Fanuc TP program (LS listing): ground_truth.ls

/PROG  TOR_XL_LEARN_V3
/ATTR
OWNER		= MNEDITOR;
COMMENT		= "WeldPRO Auto-Gen";
PROG_SIZE	= 7125;
CREATE		= DATE 26-07-30  TIME 15:09:28;
MODIFIED	= DATE 26-07-30  TIME 15:41:30;
FILE_NAME	= TOR_XL_L;
VERSION		= 0;
LINE_COUNT	= 113;
MEMORY_SIZE	= 7445;
PROTECT		= READ_WRITE;
TCD:  STACK_SIZE	= 0,
      TASK_PRIORITY	= 50,
      TIME_SLICE	= 0,
      BUSY_LAMP_OFF	= 0,
      ABORT_REQUEST	= 0,
      PAUSE_REQUEST	= 0;
DEFAULT_GROUP	= 1,*,*,*,*;
CONTROL_CODE	= 00000000 00000000;
/APPL
/MN
   1:  !WeldPRO Auto-Generated TPP ;
   2:  !TOR_XL_2026, TOR_xl_2907 ;
   3:   ;
   4:  UFRAME_NUM=2 ;
   5:  UTOOL_NUM=2 ;
   6:  !Feature Approach ;
   7:J P[1]{
   GP1:
	UF : 2, UT : 2,		CONFIG : 'F D T, 0, 0, 0',
	X =   924.335  mm,	Y =   780.986  mm,	Z =  -268.284  mm,
	W =  -106.495 deg,	P =   -15.000 deg,	R =    94.234 deg
};
P[2]{
   GP1:
	UF : 2, UT : 2,		CONFIG : 'F D T, 0, 0, 0',
	X =  1018.715  mm,	Y =   787.224  mm,	Z =  -235.231  mm,
	W =  -106.492 deg,	P =   -15.098 deg,	R =    90.372 deg
};
P[3]{
   GP1:
	UF : 2, UT : 2,		CONFIG : 'F D T, 0, 0, 0',
	X =  1020.495  mm,	Y =   807.281  mm,	Z =  -235.073  mm,
	W =  -106.456 deg,	P =   -15.335 deg,	R =    80.815 deg
};
P[4]{
   GP1:
	UF : 2, UT : 2,		CONFIG : 'F D T, 0, 0, 0',
	X =  1022.247  mm,	Y =   817.408  mm,	Z =  -235.756  mm,
	W =  -106.423 deg,	P =   -15.450 deg,	R =    76.090 deg
};
P[5]{
   GP1:
	UF : 2, UT : 2,		CONFIG : 'F D T, 0, 0, 0',
	X =  1025.517  mm,	Y =   826.963  mm,	Z =  -235.844  mm,
	W =  -106.378 deg,	P =   -15.565 deg,	R =    71.217 deg
};
P[6]{
   GP1:
	UF : 2, UT : 2,		CONFIG : 'F D T, 0, 0, 0',
	X =  1029.053  mm,	Y =   836.370  mm,	Z =  -235.876  mm,
	W =  -106.322 deg,	P =   -15.679 deg,	R =    66.207 deg
};
P[7]{
   GP1:
	UF : 2, UT : 2,		CONFIG : 'F D T, 0, 0, 0',
	X =  1033.689  mm,	Y =   845.357  mm,	Z =  -236.189  mm,
	W =  -106.254 deg,	P =   -15.791 deg,	R =    61.015 deg
};
P[8]{
   GP1:
	UF : 2, UT : 2,		CONFIG : 'F D T, 0, 0, 0',
	X =  1038.830  mm,	Y =   853.927  mm,	Z =  -236.142  mm,
	W =  -106.177 deg,	P =   -15.894 deg,	R =    55.979 deg
};
P[9]{
   GP1:
	UF : 2, UT : 2,		CONFIG : 'F D T, 0, 0, 0',
	X =  1045.034  mm,	Y =   861.671  mm,	Z =  -235.917  mm,
	W =  -106.096 deg,	P =   -15.986 deg,	R =    51.162 deg
};
P[10]{
   GP1:
	UF : 2, UT : 2,		CONFIG : 'F D T, 0, 0, 0',
	X =  1051.595  mm,	Y =   869.013  mm,	Z =  -235.579  mm,
	W =  -106.012 deg,	P =   -16.066 deg,	R =    46.632 deg
};
P[11]{
   GP1:
	UF : 2, UT : 2,		CONFIG : 'F D T, 0, 0, 0',
	X =  1058.405  mm,	Y =   876.388  mm,	Z =  -235.876  mm,
	W =  -105.919 deg,	P =   -16.142 deg,	R =    41.952 deg
};
P[12]{
   GP1:
	UF : 2, UT : 2,		CONFIG : 'F D T, 0, 0, 0',
	X =  1066.182  mm,	Y =   882.960  mm,	Z =  -236.508  mm,
	W =  -105.870 deg,	P =   -16.177 deg,	R =    39.609 deg
};
P[13]{
   GP1:
	UF : 2, UT : 2,		CONFIG : 'F D T, 0, 0, 0',
	X =  1074.017  mm,	Y =   888.320  mm,	Z =  -234.957  mm,
	W =  -105.777 deg,	P =   -16.235 deg,	R =    35.365 deg
};
P[14]{
   GP1:
	UF : 2, UT : 2,		CONFIG : 'F D T, 0, 0, 0',
	X =  1082.402  mm,	Y =   893.773  mm,	Z =  -235.312  mm,
	W =  -105.677 deg,	P =   -16.289 deg,	R =    30.964 deg
};
P[15]{
   GP1:
	UF : 2, UT : 2,		CONFIG : 'F D T, 0, 0, 0',
	X =  1091.030  mm,	Y =   899.008  mm,	Z =  -235.877  mm,
	W =  -105.579 deg,	P =   -16.333 deg,	R =    26.830 deg
};
P[16]{
   GP1:
	UF : 2, UT : 2,		CONFIG : 'F D T, 0, 0, 0',
	X =  1100.156  mm,	Y =   902.452  mm,	Z =  -235.103  mm,
	W =  -105.537 deg,	P =   -16.344 deg,	R =    25.018 deg
};
P[17]{
   GP1:
	UF : 2, UT : 2,		CONFIG : 'F D T, 0, 0, 0',
	X =  1109.917  mm,	Y =   906.637  mm,	Z =  -236.186  mm,
	W =  -116.027 deg,	P =   -16.063 deg,	R =    30.267 deg
};
P[18]{
   GP1:
	UF : 2, UT : 2,		CONFIG : 'F D T, 0, 0, 0',
	X =  1118.157  mm,	Y =   911.916  mm,	Z =  -235.088  mm,
	W =  -126.877 deg,	P =   -15.356 deg,	R =    25.893 deg
};
P[19]{
   GP1:
	UF : 2, UT : 2,		CONFIG : 'F D T, 0, 0, 0',
	X =  1124.146  mm,	Y =   914.820  mm,	Z =  -228.920  mm,
	W =  -119.393 deg,	P =   -15.981 deg,	R =    16.221 deg
};
P[20]{
   GP1:
	UF : 2, UT : 2,		CONFIG : 'F D T, 0, 0, 0',
	X =  1129.948  mm,	Y =   917.746  mm,	Z =  -222.103  mm,
	W =  -115.329 deg,	P =   -16.208 deg,	R =    11.788 deg
};
P[21]{
   GP1:
	UF : 2, UT : 2,		CONFIG : 'F D T, 0, 0, 0',
	X =  1135.715  mm,	Y =   919.222  mm,	Z =  -213.573  mm,
	W =  -112.639 deg,	P =   -16.315 deg,	R =     9.714 deg
};
P[22]{
   GP1:
	UF : 2, UT : 2,		CONFIG : 'F D T, 0, 0, 0',
	X =  1142.436  mm,	Y =   921.368  mm,	Z =  -205.545  mm,
	W =  -110.015 deg,	P =   -16.386 deg,	R =     9.649 deg
};
P[23]{
   GP1:
	UF : 2, UT : 2,		CONFIG : 'F D T, 0, 0, 0',
	X =  1147.023  mm,	Y =   921.905  mm,	Z =  -202.145  mm,
	W =  -108.552 deg,	P =   -16.418 deg,	R =     8.950 deg
};
P[24]{
   GP1:
	UF : 2, UT : 2,		CONFIG : 'F D T, 0, 0, 0',
	X =  1160.278  mm,	Y =   924.170  mm,	Z =  -197.796  mm,
	W =  -105.409 deg,	P =   -16.443 deg,	R =     6.805 deg
};
P[25]{
   GP1:
	UF : 2, UT : 2,		CONFIG : 'F D T, 0, 0, 0',
	X =  1169.888  mm,	Y =   925.126  mm,	Z =  -196.732  mm,
	W =  -104.866 deg,	P =   -16.444 deg,	R =     5.597 deg
};
P[26]{
   GP1:
	UF : 2, UT : 2,		CONFIG : 'F D T, 0, 0, 0',
	X =  1179.662  mm,	Y =   926.011  mm,	Z =  -196.715  mm,
	W =  -104.887 deg,	P =   -16.444 deg,	R =     3.523 deg
};
P[27]{
   GP1:
	UF : 2, UT : 2,		CONFIG : 'F D T, 0, 0, 0',
	X =  1189.383  mm,	Y =   926.437  mm,	Z =  -196.950  mm,
	W =  -104.930 deg,	P =   -16.439 deg,	R =     -.729 deg
};
P[28]{
   GP1:
	UF : 2, UT : 2,		CONFIG : 'F D T, 0, 0, 0',
	X =  1199.044  mm,	Y =   925.579  mm,	Z =  -197.248  mm,
	W =  -104.979 deg,	P =   -16.424 deg,	R =    -5.541 deg
};
P[29]{
   GP1:
	UF : 2, UT : 2,		CONFIG : 'F D T, 0, 0, 0',
	X =  1208.438  mm,	Y =   924.247  mm,	Z =  -196.868  mm,
	W =  -105.028 deg,	P =   -16.400 deg,	R =   -10.259 deg
};
P[30]{
   GP1:
	UF : 2, UT : 2,		CONFIG : 'F D T, 0, 0, 0',
	X =  1218.046  mm,	Y =   922.651  mm,	Z =  -197.246  mm,
	W =  -105.070 deg,	P =   -16.371 deg,	R =   -14.490 deg
};
P[31]{
   GP1:
	UF : 2, UT : 2,		CONFIG : 'F D T, 0, 0, 0',
	X =  1227.367  mm,	Y =   919.386  mm,	Z =  -197.752  mm,
	W =  -105.112 deg,	P =   -16.334 deg,	R =   -18.515 deg
};
P[32]{
   GP1:
	UF : 2, UT : 2,		CONFIG : 'F D T, 0, 0, 0',
	X =  1236.641  mm,	Y =   916.419  mm,	Z =  -198.075  mm,
	W =  -105.158 deg,	P =   -16.285 deg,	R =   -23.051 deg
};
P[33]{
   GP1:
	UF : 2, UT : 2,		CONFIG : 'F D T, 0, 0, 0',
	X =  1245.126  mm,	Y =   912.315  mm,	Z =  -197.759  mm,
	W =  -105.219 deg,	P =   -16.204 deg,	R =   -29.417 deg
};
P[34]{
   GP1:
	UF : 2, UT : 2,		CONFIG : 'F D T, 0, 0, 0',
	X =  1252.682  mm,	Y =   907.045  mm,	Z =  -197.652  mm,
	W =  -105.311 deg,	P =   -16.047 deg,	R =   -39.415 deg
};
P[35]{
   GP1:
	UF : 2, UT : 2,		CONFIG : 'F D T, 0, 0, 0',
	X =  1260.941  mm,	Y =   901.305  mm,	Z =  -197.740  mm,
	W =  -105.307 deg,	P =   -16.055 deg,	R =   -38.974 deg
};
P[36]{
   GP1:
	UF : 2, UT : 2,		CONFIG : 'F D T, 0, 0, 0',
	X =  1267.955  mm,	Y =   894.273  mm,	Z =  -197.409  mm,
	W =  -105.302 deg,	P =   -16.063 deg,	R =   -38.625 deg
};
P[37]{
   GP1:
	UF : 2, UT : 2,		CONFIG : 'F D T, 0, 0, 0',
	X =  1276.534  mm,	Y =   889.263  mm,	Z =  -197.995  mm,
	W =  -105.469 deg,	P =   -15.944 deg,	R =   -44.976 deg
};
P[38]{
   GP1:
	UF : 2, UT : 2,		CONFIG : 'F D T, 0, 0, 0',
	X =  1283.155  mm,	Y =   882.295  mm,	Z =  -197.847  mm,
	W =  -105.661 deg,	P =   -15.890 deg,	R =   -47.714 deg
};
P[39]{
   GP1:
	UF : 2, UT : 2,		CONFIG : 'F D T, 0, 0, 0',
	X =  1289.852  mm,	Y =   875.249  mm,	Z =  -198.875  mm,
	W =  -106.210 deg,	P =   -15.792 deg,	R =   -52.259 deg
};
P[40]{
   GP1:
	UF : 2, UT : 2,		CONFIG : 'F D T, 0, 0, 0',
	X =  1296.112  mm,	Y =   867.768  mm,	Z =  -200.273  mm,
	W =  -106.927 deg,	P =   -15.688 deg,	R =   -56.663 deg
};
P[41]{
   GP1:
	UF : 2, UT : 2,		CONFIG : 'F D T, 0, 0, 0',
	X =  1301.774  mm,	Y =   859.713  mm,	Z =  -202.128  mm,
	W =  -107.603 deg,	P =   -15.597 deg,	R =   -60.243 deg
};
P[42]{
   GP1:
	UF : 2, UT : 2,		CONFIG : 'F D T, 0, 0, 0',
	X =  1306.016  mm,	Y =   850.984  mm,	Z =  -203.650  mm,
	W =  -108.271 deg,	P =   -15.504 deg,	R =   -63.685 deg
};
P[43]{
   GP1:
	UF : 2, UT : 2,		CONFIG : 'F D T, 0, 0, 0',
	X =  1309.573  mm,	Y =   842.117  mm,	Z =  -204.775  mm,
	W =  -109.144 deg,	P =   -15.377 deg,	R =   -68.203 deg
};
P[44]{
   GP1:
	UF : 2, UT : 2,		CONFIG : 'F D T, 0, 0, 0',
	X =  1313.875  mm,	Y =   833.270  mm,	Z =  -206.451  mm,
	W =  -109.899 deg,	P =   -15.253 deg,	R =   -72.505 deg
};
P[45]{
   GP1:
	UF : 2, UT : 2,		CONFIG : 'F D T, 0, 0, 0',
	X =  1317.383  mm,	Y =   823.850  mm,	Z =  -208.446  mm,
	W =  -110.273 deg,	P =   -15.181 deg,	R =   -74.981 deg
};
P[46]{
   GP1:
	UF : 2, UT : 2,		CONFIG : 'F D T, 0, 0, 0',
	X =  1319.294  mm,	Y =   814.046  mm,	Z =  -209.598  mm,
	W =  -110.635 deg,	P =   -14.305 deg,	R =   -78.232 deg
};
P[47]{
   GP1:
	UF : 2, UT : 2,		CONFIG : 'F D T, 0, 0, 0',
	X =  1321.222  mm,	Y =   804.155  mm,	Z =  -210.895  mm,
	W =  -111.054 deg,	P =   -14.769 deg,	R =   -83.164 deg
};
P[48]{
   GP1:
	UF : 2, UT : 2,		CONFIG : 'F D T, 0, 0, 0',
	X =  1322.108  mm,	Y =   794.074  mm,	Z =  -211.690  mm,
	W =  -111.190 deg,	P =   -15.305 deg,	R =   -88.308 deg
};
P[49]{
   GP1:
	UF : 2, UT : 2,		CONFIG : 'F D T, 0, 0, 0',
	X =  1322.417  mm,	Y =   783.924  mm,	Z =  -211.983  mm,
	W =  -111.129 deg,	P =   -15.645 deg,	R =   -91.614 deg
};
P[50]{
   GP1:
	UF : 2, UT : 2,		CONFIG : 'F D T, 0, 0, 0',
	X =  1321.632  mm,	Y =   773.848  mm,	Z =  -211.329  mm,
	W =  -110.761 deg,	P =   -14.624 deg,	R =   -96.574 deg
};
P[51]{
   GP1:
	UF : 2, UT : 2,		CONFIG : 'F D T, 0, 0, 0',
	X =  1320.812  mm,	Y =   763.757  mm,	Z =  -210.466  mm,
	W =  -110.276 deg,	P =   -14.535 deg,	R =  -100.836 deg
};
P[52]{
   GP1:
	UF : 2, UT : 2,		CONFIG : 'F D T, 0, 0, 0',
	X =  1318.396  mm,	Y =   754.196  mm,	Z =  -208.431  mm,
	W =  -109.635 deg,	P =   -14.447 deg,	R =  -105.265 deg
};
P[53]{
   GP1:
	UF : 2, UT : 2,		CONFIG : 'F D T, 0, 0, 0',
	X =  1315.879  mm,	Y =   744.538  mm,	Z =  -206.875  mm,
	W =  -109.083 deg,	P =   -14.382 deg,	R =  -108.625 deg
};
P[54]{
   GP1:
	UF : 2, UT : 2,		CONFIG : 'F D T, 0, 0, 0',
	X =  1312.567  mm,	Y =   735.090  mm,	Z =  -205.253  mm,
	W =  -108.349 deg,	P =   -14.302 deg,	R =  -112.873 deg
};
P[55]{
   GP1:
	UF : 2, UT : 2,		CONFIG : 'F D T, 0, 0, 0',
	X =  1308.961  mm,	Y =   725.703  mm,	Z =  -203.640  mm,
	W =  -107.748 deg,	P =   -14.239 deg,	R =  -116.265 deg
};
P[56]{
   GP1:
	UF : 2, UT : 2,		CONFIG : 'F D T, 0, 0, 0',
	X =  1305.001  mm,	Y =   716.454  mm,	Z =  -201.746  mm,
	W =  -106.927 deg,	P =   -14.148 deg,	R =  -121.193 deg
};
P[57]{
   GP1:
	UF : 2, UT : 2,		CONFIG : 'F D T, 0, 0, 0',
	X =  1299.050  mm,	Y =   708.363  mm,	Z =  -199.926  mm,
	W =  -106.269 deg,	P =   -14.066 deg,	R =  -125.698 deg
};
P[58]{
   GP1:
	UF : 2, UT : 2,		CONFIG : 'F D T, 0, 0, 0',
	X =  1293.324  mm,	Y =   700.186  mm,	Z =  -198.073  mm,
	W =  -105.781 deg,	P =   -13.988 deg,	R =  -130.143 deg
};
P[59]{
   GP1:
	UF : 2, UT : 2,		CONFIG : 'F D T, 0, 0, 0',
	X =  1286.894  mm,	Y =   692.340  mm,	Z =  -197.040  mm,
	W =  -105.529 deg,	P =   -13.914 deg,	R =  -134.519 deg
};
P[60]{
   GP1:
	UF : 2, UT : 2,		CONFIG : 'F D T, 0, 0, 0',
	X =  1279.894  mm,	Y =   684.848  mm,	Z =  -196.766  mm,
	W =  -105.437 deg,	P =   -13.849 deg,	R =  -138.629 deg
};
P[61]{
   GP1:
	UF : 2, UT : 2,		CONFIG : 'F D T, 0, 0, 0',
	X =  1272.475  mm,	Y =   678.006  mm,	Z =  -196.723  mm,
	W =  -105.429 deg,	P =   -13.831 deg,	R =  -139.837 deg
};
P[62]{
   GP1:
	UF : 2, UT : 2,		CONFIG : 'F D T, 0, 0, 0',
	X =  1265.641  mm,	Y =   670.880  mm,	Z =  -196.694  mm,
	W =  -105.443 deg,	P =   -13.863 deg,	R =  -137.727 deg
};
P[63]{
   GP1:
	UF : 2, UT : 2,		CONFIG : 'F D T, 0, 0, 0',
	X =  1257.021  mm,	Y =   664.482  mm,	Z =  -196.380  mm,
	W =  -105.373 deg,	P =   -13.729 deg,	R =  -147.436 deg
};
P[64]{
   GP1:
	UF : 2, UT : 2,		CONFIG : 'F D T, 0, 0, 0',
	X =  1247.675  mm,	Y =   659.504  mm,	Z =  -196.028  mm,
	W =  -105.298 deg,	P =   -13.637 deg,	R =  -156.529 deg
};
P[65]{
   GP1:
	UF : 2, UT : 2,		CONFIG : 'F D T, 0, 0, 0',
	X =  1238.718  mm,	Y =   654.671  mm,	Z =  -195.720  mm,
	W =  -105.277 deg,	P =   -13.618 deg,	R =  -158.976 deg
};
P[66]{
   GP1:
	UF : 2, UT : 2,		CONFIG : 'F D T, 0, 0, 0',
	X =  1229.052  mm,	Y =   650.811  mm,	Z =  -195.862  mm,
	W =  -105.241 deg,	P =   -13.592 deg,	R =  -162.969 deg
};
P[67]{
   GP1:
	UF : 2, UT : 2,		CONFIG : 'F D T, 0, 0, 0',
	X =  1219.160  mm,	Y =   648.075  mm,	Z =  -195.385  mm,
	W =  -105.203 deg,	P =   -13.573 deg,	R =  -167.022 deg
};
P[68]{
   GP1:
	UF : 2, UT : 2,		CONFIG : 'F D T, 0, 0, 0',
	X =  1208.921  mm,	Y =   646.203  mm,	Z =  -195.395  mm,
	W =  -105.159 deg,	P =   -13.560 deg,	R =  -171.569 deg
};
P[69]{
   GP1:
	UF : 2, UT : 2,		CONFIG : 'F D T, 0, 0, 0',
	X =  1198.642  mm,	Y =   645.785  mm,	Z =  -194.956  mm,
	W =  -105.113 deg,	P =   -13.556 deg,	R =  -176.312 deg
};
P[70]{
   GP1:
	UF : 2, UT : 2,		CONFIG : 'F D T, 0, 0, 0',
	X =  1188.344  mm,	Y =   645.393  mm,	Z =  -194.871  mm,
	W =  -105.068 deg,	P =   -13.561 deg,	R =   179.213 deg
};
P[71]{
   GP1:
	UF : 2, UT : 2,		CONFIG : 'F D T, 0, 0, 0',
	X =  1178.059  mm,	Y =   645.736  mm,	Z =  -195.139  mm,
	W =  -105.038 deg,	P =   -13.569 deg,	R =   176.231 deg
};
P[72]{
   GP1:
	UF : 2, UT : 2,		CONFIG : 'F D T, 0, 0, 0',
	X =  1167.871  mm,	Y =   646.652  mm,	Z =  -195.801  mm,
	W =  -105.207 deg,	P =   -13.572 deg,	R =   175.290 deg
};
P[73]{
   GP1:
	UF : 2, UT : 2,		CONFIG : 'F D T, 0, 0, 0',
	X =  1158.477  mm,	Y =   647.343  mm,	Z =  -195.653  mm,
	W =  -107.012 deg,	P =   -13.569 deg,	R =   174.537 deg
};
P[74]{
   GP1:
	UF : 2, UT : 2,		CONFIG : 'F D T, 0, 0, 0',
	X =  1149.730  mm,	Y =   648.837  mm,	Z =  -198.834  mm,
	W =  -109.414 deg,	P =   -13.538 deg,	R =   174.483 deg
};
P[75]{
   GP1:
	UF : 2, UT : 2,		CONFIG : 'F D T, 0, 0, 0',
	X =  1141.667  mm,	Y =   649.097  mm,	Z =  -206.147  mm,
	W =  -112.196 deg,	P =   -13.466 deg,	R =   175.323 deg
};
P[76]{
   GP1:
	UF : 2, UT : 2,		CONFIG : 'F D T, 0, 0, 0',
	X =  1135.547  mm,	Y =   650.958  mm,	Z =  -213.092  mm,
	W =  -114.872 deg,	P =   -13.369 deg,	R =   175.422 deg
};
P[77]{
   GP1:
	UF : 2, UT : 2,		CONFIG : 'F D T, 0, 0, 0',
	X =  1128.794  mm,	Y =   652.546  mm,	Z =  -221.828  mm,
	W =  -120.114 deg,	P =   -13.109 deg,	R =   172.293 deg
};
P[78]{
   GP1:
	UF : 2, UT : 2,		CONFIG : 'F D T, 0, 0, 0',
	X =  1122.507  mm,	Y =   656.297  mm,	Z =  -228.913  mm,
	W =  -126.810 deg,	P =   -12.622 deg,	R =   167.787 deg
};
P[79]{
   GP1:
	UF : 2, UT : 2,		CONFIG : 'F D T, 0, 0, 0',
	X =  1113.925  mm,	Y =   660.943  mm,	Z =  -232.976  mm,
	W =  -119.561 deg,	P =   -13.285 deg,	R =   157.806 deg
};
P[80]{
   GP1:
	UF : 2, UT : 2,		CONFIG : 'F D T, 0, 0, 0',
	X =  1104.936  mm,	Y =   665.580  mm,	Z =  -233.167  mm,
	W =  -107.219 deg,	P =   -13.741 deg,	R =   154.408 deg
};
P[81]{
   GP1:
	UF : 2, UT : 2,		CONFIG : 'F D T, 0, 0, 0',
	X =  1095.534  mm,	Y =   669.254  mm,	Z =  -233.425  mm,
	W =  -105.746 deg,	P =   -13.749 deg,	R =   154.142 deg
};
P[82]{
   GP1:
	UF : 2, UT : 2,		CONFIG : 'F D T, 0, 0, 0',
	X =  1086.430  mm,	Y =   673.774  mm,	Z =  -233.281  mm,
	W =  -105.804 deg,	P =   -13.784 deg,	R =   151.506 deg
};
P[83]{
   GP1:
	UF : 2, UT : 2,		CONFIG : 'F D T, 0, 0, 0',
	X =  1077.665  mm,	Y =   679.493  mm,	Z =  -233.931  mm,
	W =  -105.885 deg,	P =   -13.838 deg,	R =   147.739 deg
};
P[84]{
   GP1:
	UF : 2, UT : 2,		CONFIG : 'F D T, 0, 0, 0',
	X =  1069.342  mm,	Y =   685.844  mm,	Z =  -234.331  mm,
	W =  -105.988 deg,	P =   -13.918 deg,	R =   142.681 deg
};
P[85]{
   GP1:
	UF : 2, UT : 2,		CONFIG : 'F D T, 0, 0, 0',
	X =  1061.489  mm,	Y =   692.528  mm,	Z =  -234.339  mm,
	W =  -106.082 deg,	P =   -14.006 deg,	R =   137.688 deg
};
P[86]{
   GP1:
	UF : 2, UT : 2,		CONFIG : 'F D T, 0, 0, 0',
	X =  1054.334  mm,	Y =   699.587  mm,	Z =  -234.035  mm,
	W =  -106.129 deg,	P =   -14.056 deg,	R =   135.015 deg
};
P[87]{
   GP1:
	UF : 2, UT : 2,		CONFIG : 'F D T, 0, 0, 0',
	X =  1046.717  mm,	Y =   706.698  mm,	Z =  -234.774  mm,
	W =  -106.186 deg,	P =   -14.117 deg,	R =   131.622 deg
};
P[88]{
   GP1:
	UF : 2, UT : 2,		CONFIG : 'F D T, 0, 0, 0',
	X =  1040.975  mm,	Y =   715.201  mm,	Z =  -234.549  mm,
	W =  -106.269 deg,	P =   -14.239 deg,	R =   125.999 deg
};
P[89]{
   GP1:
	UF : 2, UT : 2,		CONFIG : 'F D T, 0, 0, 0',
	X =  1035.094  mm,	Y =   723.442  mm,	Z =  -234.529  mm,
	W =  -106.343 deg,	P =   -14.367 deg,	R =   120.225 deg
};
P[90]{
   GP1:
	UF : 2, UT : 2,		CONFIG : 'F D T, 0, 0, 0',
	X =  1030.109  mm,	Y =   732.680  mm,	Z =  -235.085  mm,
	W =  -106.384 deg,	P =   -14.458 deg,	R =   116.261 deg
};
P[91]{
   GP1:
	UF : 2, UT : 2,		CONFIG : 'F D T, 0, 0, 0',
	X =  1027.450  mm,	Y =   740.213  mm,	Z =  -234.571  mm,
	W =  -106.433 deg,	P =   -14.556 deg,	R =   111.957 deg
};
P[92]{
   GP1:
	UF : 2, UT : 2,		CONFIG : 'F D T, 0, 0, 0',
	X =  1023.176  mm,	Y =   751.884  mm,	Z =  -234.975  mm,
	W =  -106.465 deg,	P =   -14.714 deg,	R =   105.666 deg
};
P[93]{
   GP1:
	UF : 2, UT : 2,		CONFIG : 'F D T, 0, 1, 0',
	X =  1021.222  mm,	Y =   761.846  mm,	Z =  -235.095  mm,
	W =  -106.480 deg,	P =   -14.798 deg,	R =   102.262 deg
};
P[94]{
   GP1:
	UF : 2, UT : 2,		CONFIG : 'F D T, 0, 1, 0',
	X =  1019.798  mm,	Y =   771.823  mm,	Z =  -234.842  mm,
	W =  -106.494 deg,	P =   -14.935 deg,	R =    96.827 deg
};
P[95]{
   GP1:
	UF : 2, UT : 2,		CONFIG : 'F D T, 0, 0, 0',
	X =  1018.674  mm,	Y =   779.059  mm,	Z =  -235.046  mm,
	W =  -106.499 deg,	P =   -14.997 deg,	R =    94.225 deg
};
P[96]{
   GP1:
	UF : 2, UT : 2,		CONFIG : 'F D T, 0, 1, 0',
	X =  1018.425  mm,	Y =   779.122  mm,	Z =  -235.344  mm,
	W =  -106.501 deg,	P =   -14.999 deg,	R =    94.236 deg
};
P[97]{
   GP1:
	UF : 2, UT : 2,		CONFIG : 'F D T, 0, 0, 0',
	X =  1018.875  mm,	Y =   797.394  mm,	Z =  -235.383  mm,
	W =  -106.481 deg,	P =   -15.218 deg,	R =    85.605 deg
};
P[98]{
   GP1:
	UF : 2, UT : 2,		CONFIG : 'F D T, 0, 1, 0',
	X =   651.995  mm,	Y =   781.694  mm,	Z =  -345.952  mm,
	W =  -106.495 deg,	P =   -15.000 deg,	R =    94.234 deg
};

/END
